// Mitsubishi GX Works2 project: AUTOROLLING_3073_6_2_2026   PLC: Q06UDV
// AUTOROLLING_3073_6_2_2024

PROGRAM 01
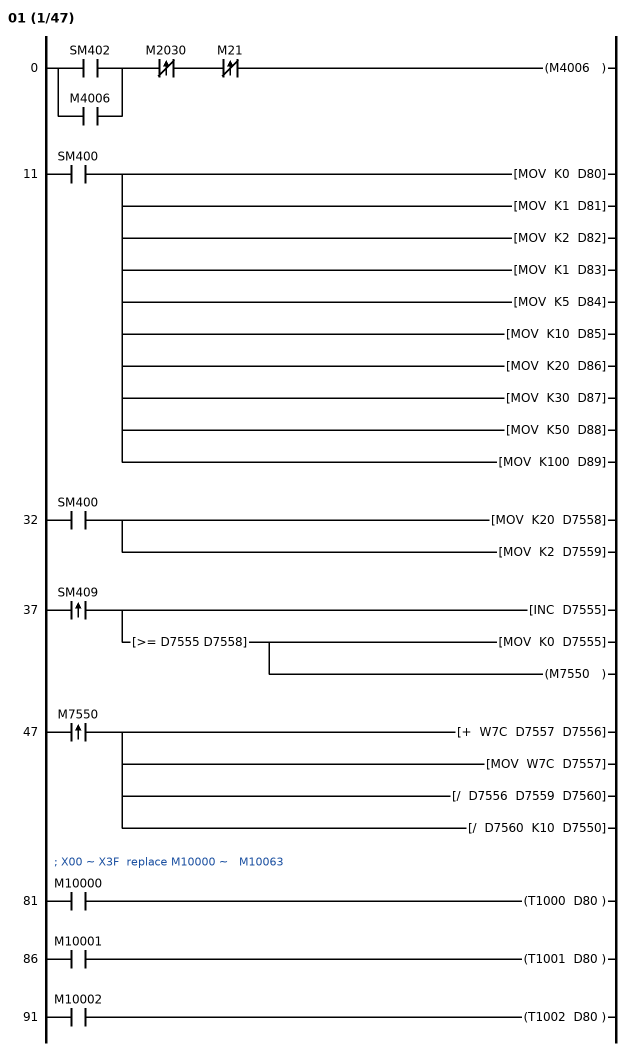
0     LD      SM402
      OR      M4006
      ANDPI   M2030
      ANDPI   M21
      OUT     M4006
; 
; 
; 
11    LD      SM400
      MOV     K0 D80
      MOV     K1 D81
      MOV     K2 D82
      MOV     K1 D83
      MOV     K5 D84
      MOV     K10 D85
      MOV     K20 D86
      MOV     K30 D87
      MOV     K50 D88
      MOV     K100 D89
32    LD      SM400
      MOV     K20 D7558
      MOV     K2 D7559
37    LDP     SM409
      INC     D7555
      AND>=   D7555 D7558
      MOV     K0 D7555
      OUT     M7550
47    LDP     M7550
      +       W7C D7557 D7556
      MOV     W7C D7557
      /       D7556 D7559 D7560
      /       D7560 K10 D7550
; X00 ~ X3F  replace M10000 ~　M10063
81    LD      M10000
      OUT     T1000 D80
86    LD      M10001
      OUT     T1001 D80
91    LD      M10002
      OUT     T1002 D80
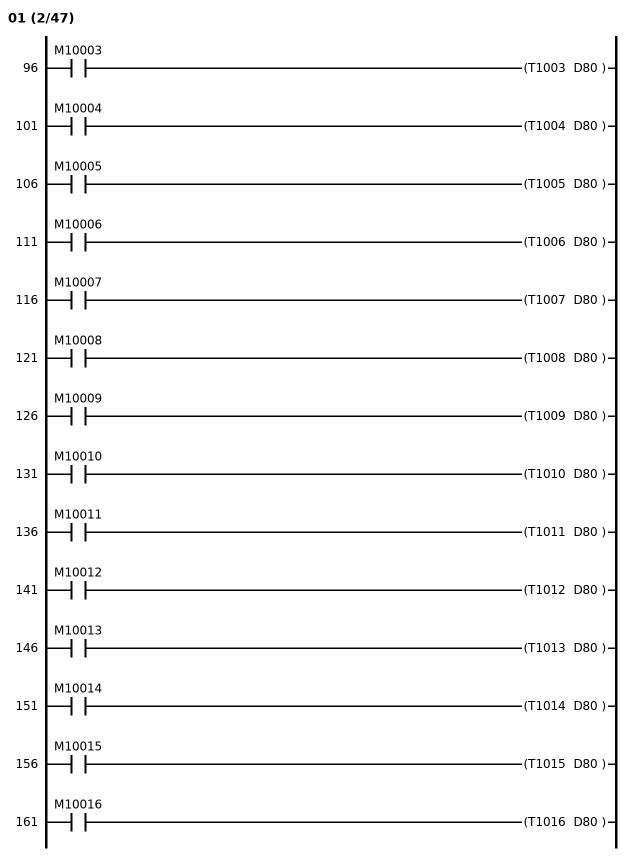
96    LD      M10003
      OUT     T1003 D80
101   LD      M10004
      OUT     T1004 D80
106   LD      M10005
      OUT     T1005 D80
111   LD      M10006
      OUT     T1006 D80
116   LD      M10007
      OUT     T1007 D80
121   LD      M10008
      OUT     T1008 D80
126   LD      M10009
      OUT     T1009 D80
131   LD      M10010
      OUT     T1010 D80
136   LD      M10011
      OUT     T1011 D80
141   LD      M10012
      OUT     T1012 D80
146   LD      M10013
      OUT     T1013 D80
151   LD      M10014
      OUT     T1014 D80
156   LD      M10015
      OUT     T1015 D80
161   LD      M10016
      OUT     T1016 D80
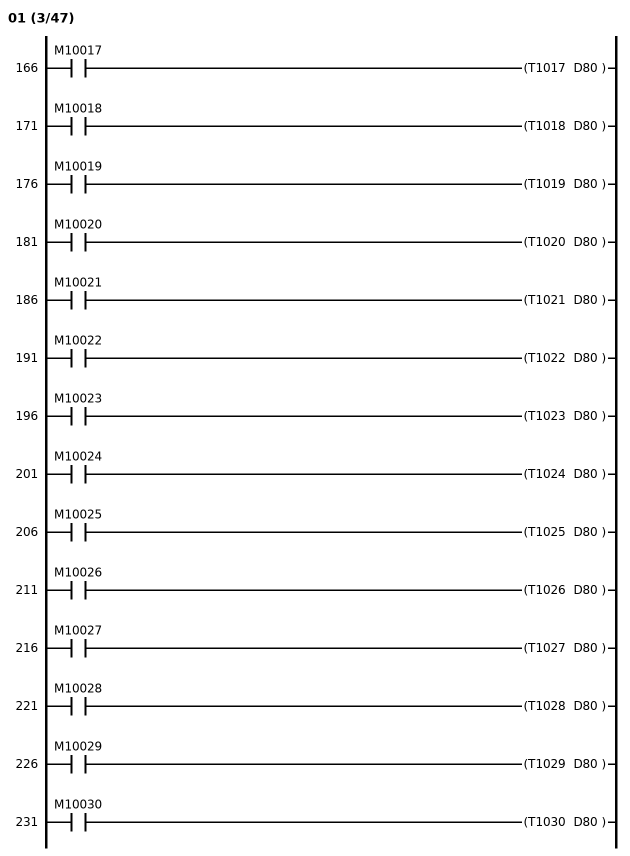
166   LD      M10017
      OUT     T1017 D80
171   LD      M10018
      OUT     T1018 D80
176   LD      M10019
      OUT     T1019 D80
181   LD      M10020
      OUT     T1020 D80
186   LD      M10021
      OUT     T1021 D80
191   LD      M10022
      OUT     T1022 D80
196   LD      M10023
      OUT     T1023 D80
201   LD      M10024
      OUT     T1024 D80
206   LD      M10025
      OUT     T1025 D80
211   LD      M10026
      OUT     T1026 D80
216   LD      M10027
      OUT     T1027 D80
221   LD      M10028
      OUT     T1028 D80
226   LD      M10029
      OUT     T1029 D80
231   LD      M10030
      OUT     T1030 D80
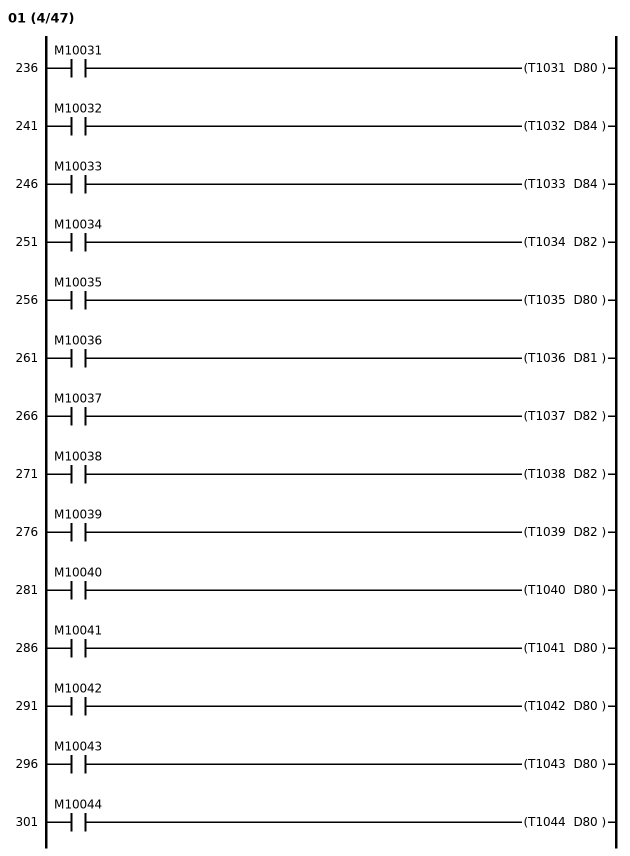
236   LD      M10031
      OUT     T1031 D80
241   LD      M10032
      OUT     T1032 D84
246   LD      M10033
      OUT     T1033 D84
251   LD      M10034
      OUT     T1034 D82
256   LD      M10035
      OUT     T1035 D80
261   LD      M10036
      OUT     T1036 D81
266   LD      M10037
      OUT     T1037 D82
271   LD      M10038
      OUT     T1038 D82
276   LD      M10039
      OUT     T1039 D82
281   LD      M10040
      OUT     T1040 D80
286   LD      M10041
      OUT     T1041 D80
291   LD      M10042
      OUT     T1042 D80
296   LD      M10043
      OUT     T1043 D80
301   LD      M10044
      OUT     T1044 D80
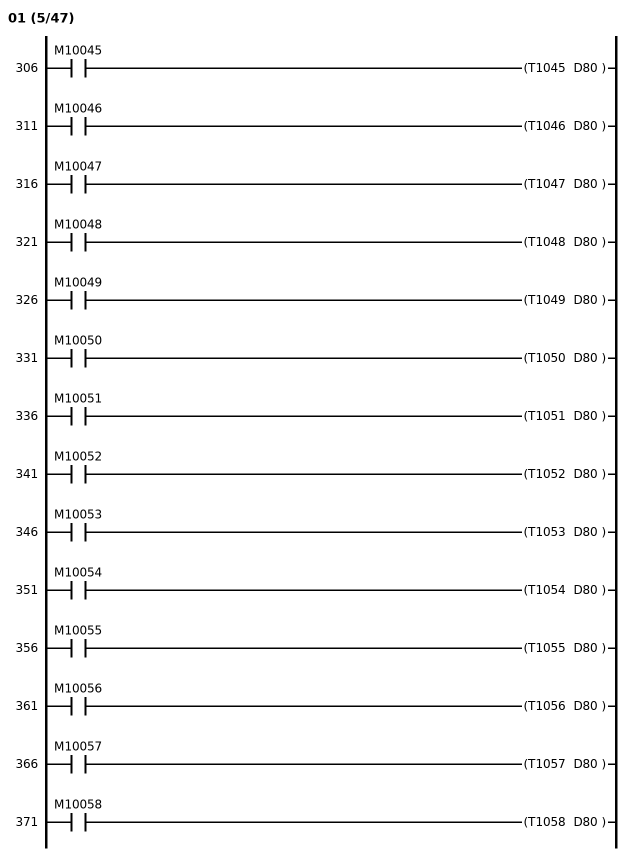
306   LD      M10045
      OUT     T1045 D80
311   LD      M10046
      OUT     T1046 D80
316   LD      M10047
      OUT     T1047 D80
321   LD      M10048
      OUT     T1048 D80
326   LD      M10049
      OUT     T1049 D80
331   LD      M10050
      OUT     T1050 D80
336   LD      M10051
      OUT     T1051 D80
341   LD      M10052
      OUT     T1052 D80
346   LD      M10053
      OUT     T1053 D80
351   LD      M10054
      OUT     T1054 D80
356   LD      M10055
      OUT     T1055 D80
361   LD      M10056
      OUT     T1056 D80
366   LD      M10057
      OUT     T1057 D80
371   LD      M10058
      OUT     T1058 D80
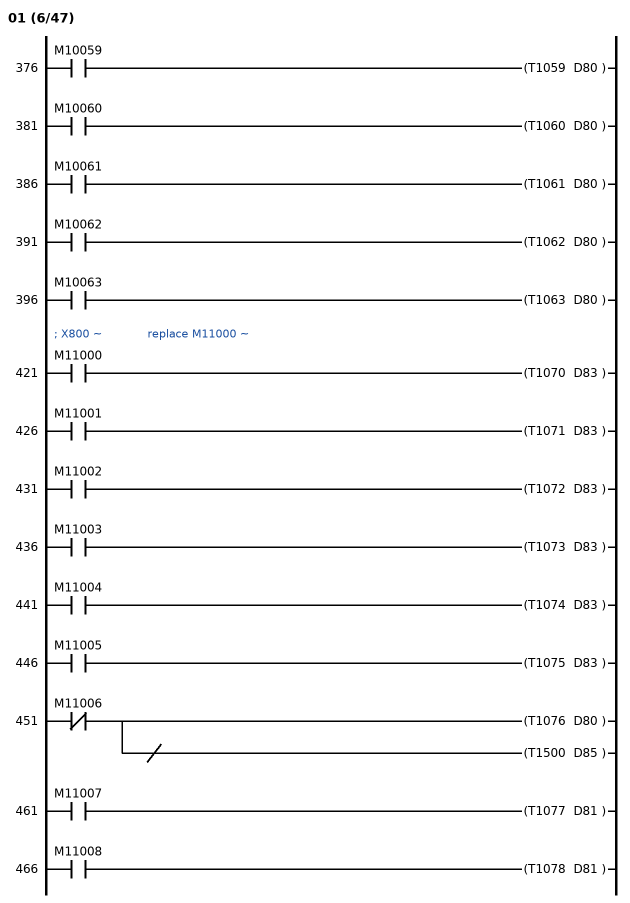
376   LD      M10059
      OUT     T1059 D80
381   LD      M10060
      OUT     T1060 D80
386   LD      M10061
      OUT     T1061 D80
391   LD      M10062
      OUT     T1062 D80
396   LD      M10063
      OUT     T1063 D80
; X800 ~             replace M11000 ~
421   LD      M11000
      OUT     T1070 D83
426   LD      M11001
      OUT     T1071 D83
431   LD      M11002
      OUT     T1072 D83
436   LD      M11003
      OUT     T1073 D83
441   LD      M11004
      OUT     T1074 D83
446   LD      M11005
      OUT     T1075 D83
451   LDI     M11006
      OUT     T1076 D80
      INV
      OUT     T1500 D85
461   LD      M11007
      OUT     T1077 D81
466   LD      M11008
      OUT     T1078 D81
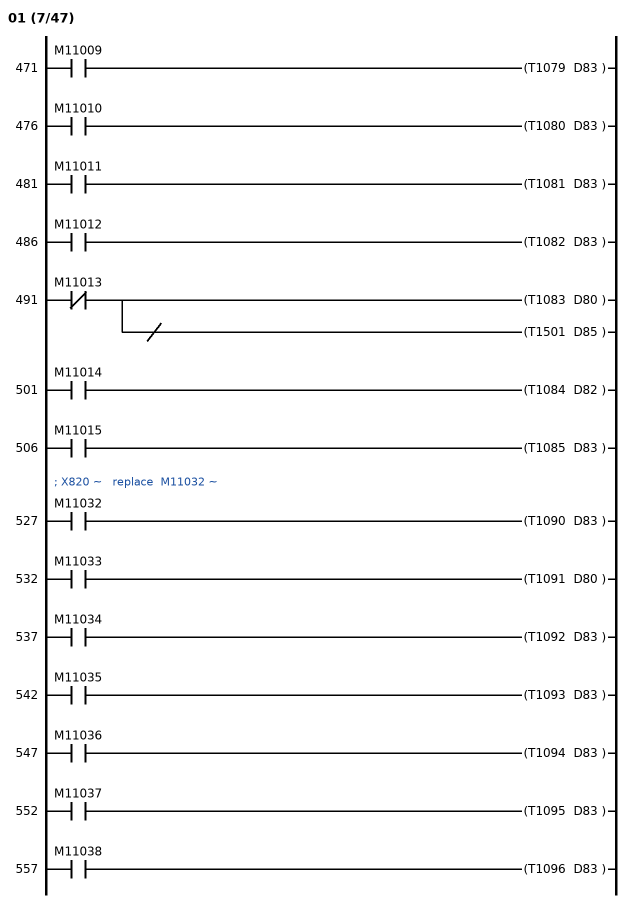
471   LD      M11009
      OUT     T1079 D83
476   LD      M11010
      OUT     T1080 D83
481   LD      M11011
      OUT     T1081 D83
486   LD      M11012
      OUT     T1082 D83
491   LDI     M11013
      OUT     T1083 D80
      INV
      OUT     T1501 D85
501   LD      M11014
      OUT     T1084 D82
506   LD      M11015
      OUT     T1085 D83
; X820 ~   replace  M11032 ~
527   LD      M11032
      OUT     T1090 D83
532   LD      M11033
      OUT     T1091 D80
537   LD      M11034
      OUT     T1092 D83
542   LD      M11035
      OUT     T1093 D83
547   LD      M11036
      OUT     T1094 D83
552   LD      M11037
      OUT     T1095 D83
557   LD      M11038
      OUT     T1096 D83
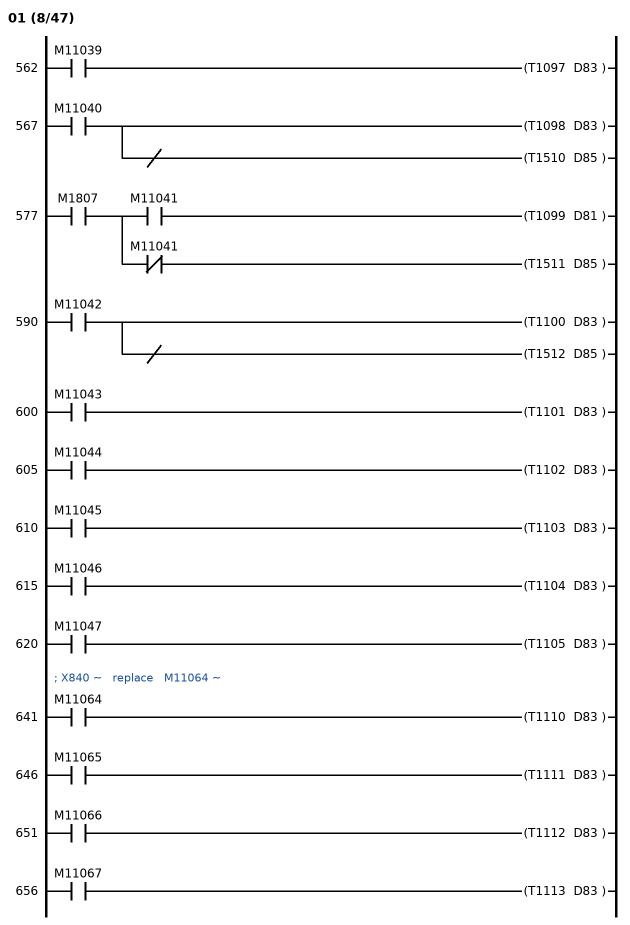
562   LD      M11039
      OUT     T1097 D83
567   LD      M11040
      OUT     T1098 D83
      INV
      OUT     T1510 D85
577   LD      M1807
      MPS
      AND     M11041
      OUT     T1099 D81
      MPP
      ANI     M11041
      OUT     T1511 D85
590   LD      M11042
      OUT     T1100 D83
      INV
      OUT     T1512 D85
600   LD      M11043
      OUT     T1101 D83
605   LD      M11044
      OUT     T1102 D83
610   LD      M11045
      OUT     T1103 D83
615   LD      M11046
      OUT     T1104 D83
620   LD      M11047
      OUT     T1105 D83
; X840 ~   replace   M11064 ~
641   LD      M11064
      OUT     T1110 D83
646   LD      M11065
      OUT     T1111 D83
651   LD      M11066
      OUT     T1112 D83
656   LD      M11067
      OUT     T1113 D83
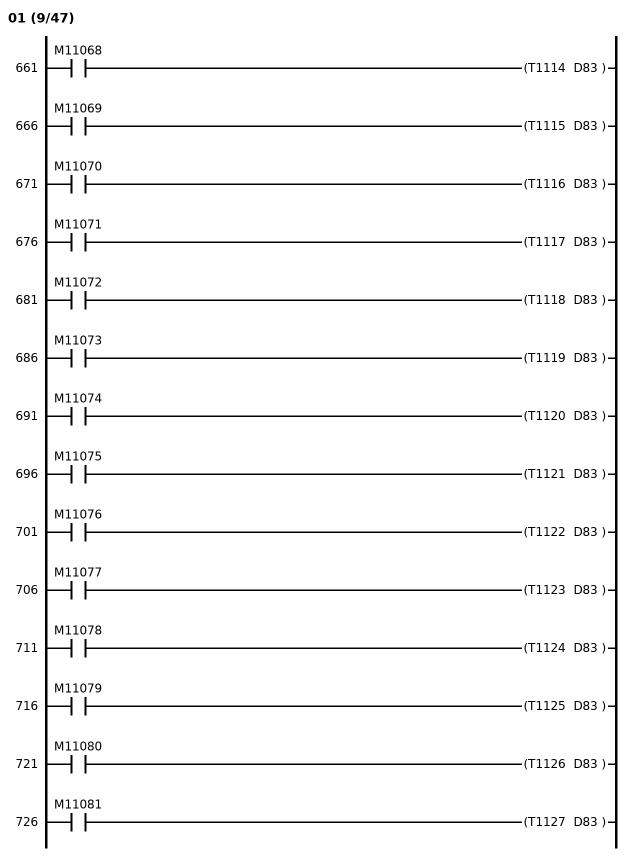
661   LD      M11068
      OUT     T1114 D83
666   LD      M11069
      OUT     T1115 D83
671   LD      M11070
      OUT     T1116 D83
676   LD      M11071
      OUT     T1117 D83
681   LD      M11072
      OUT     T1118 D83
686   LD      M11073
      OUT     T1119 D83
691   LD      M11074
      OUT     T1120 D83
696   LD      M11075
      OUT     T1121 D83
701   LD      M11076
      OUT     T1122 D83
706   LD      M11077
      OUT     T1123 D83
711   LD      M11078
      OUT     T1124 D83
716   LD      M11079
      OUT     T1125 D83
721   LD      M11080
      OUT     T1126 D83
726   LD      M11081
      OUT     T1127 D83
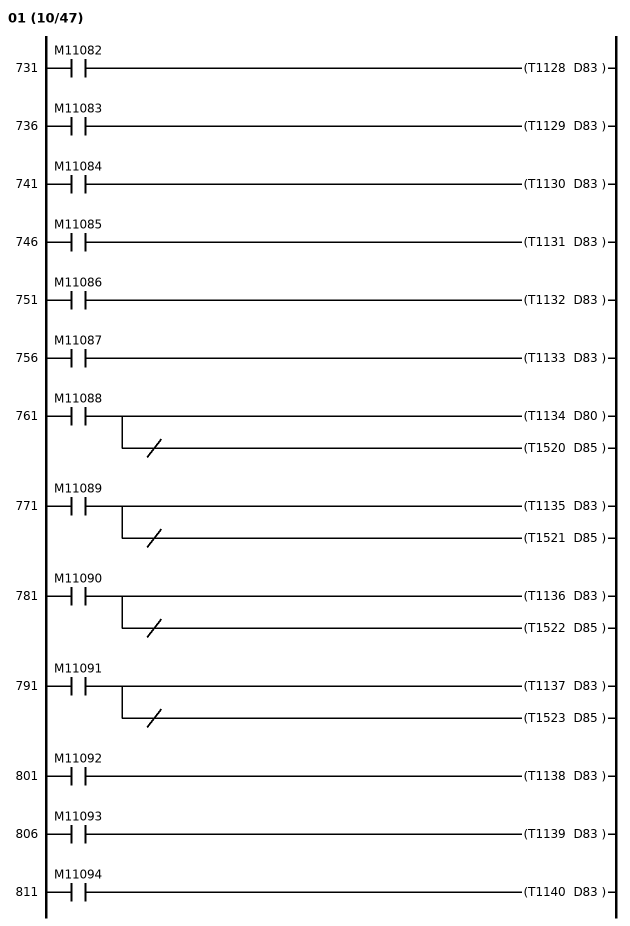
731   LD      M11082
      OUT     T1128 D83
736   LD      M11083
      OUT     T1129 D83
741   LD      M11084
      OUT     T1130 D83
746   LD      M11085
      OUT     T1131 D83
751   LD      M11086
      OUT     T1132 D83
756   LD      M11087
      OUT     T1133 D83
761   LD      M11088
      OUT     T1134 D80
      INV
      OUT     T1520 D85
771   LD      M11089
      OUT     T1135 D83
      INV
      OUT     T1521 D85
781   LD      M11090
      OUT     T1136 D83
      INV
      OUT     T1522 D85
791   LD      M11091
      OUT     T1137 D83
      INV
      OUT     T1523 D85
801   LD      M11092
      OUT     T1138 D83
806   LD      M11093
      OUT     T1139 D83
811   LD      M11094
      OUT     T1140 D83
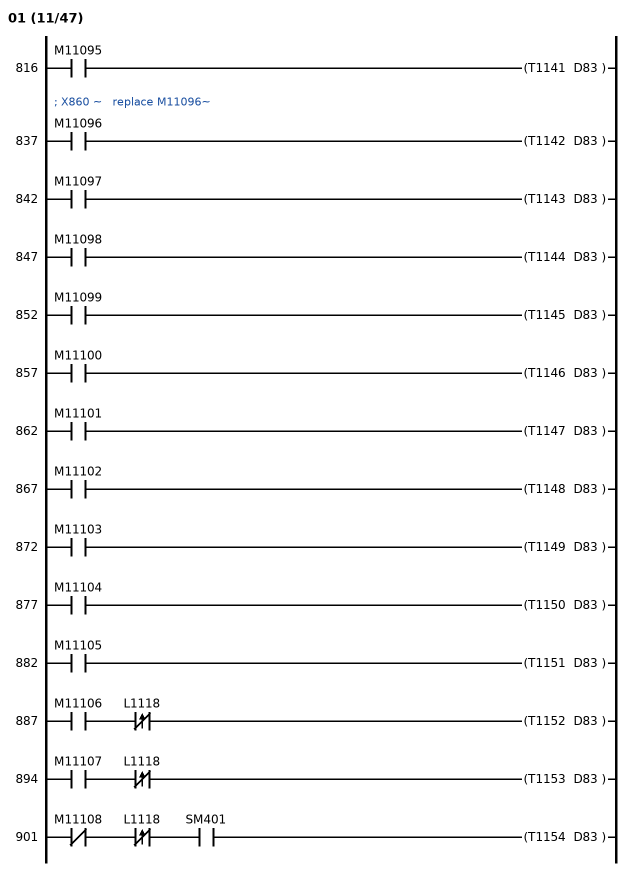
816   LD      M11095
      OUT     T1141 D83
; X860 ~   replace M11096~
837   LD      M11096
      OUT     T1142 D83
842   LD      M11097
      OUT     T1143 D83
847   LD      M11098
      OUT     T1144 D83
852   LD      M11099
      OUT     T1145 D83
857   LD      M11100
      OUT     T1146 D83
862   LD      M11101
      OUT     T1147 D83
867   LD      M11102
      OUT     T1148 D83
872   LD      M11103
      OUT     T1149 D83
877   LD      M11104
      OUT     T1150 D83
882   LD      M11105
      OUT     T1151 D83
887   LD      M11106
      ANDPI   L1118
      OUT     T1152 D83
894   LD      M11107
      ANDPI   L1118
      OUT     T1153 D83
901   LDI     M11108
      ANDPI   L1118
      AND     SM401
      OUT     T1154 D83
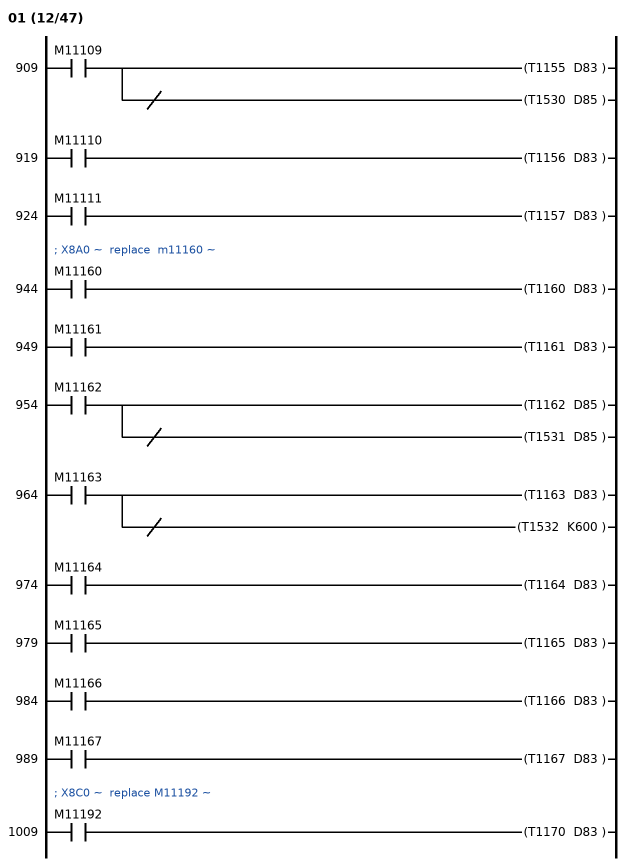
909   LD      M11109
      OUT     T1155 D83
      INV
      OUT     T1530 D85
919   LD      M11110
      OUT     T1156 D83
924   LD      M11111
      OUT     T1157 D83
; X8A0 ~  replace  m11160 ~
944   LD      M11160
      OUT     T1160 D83
949   LD      M11161
      OUT     T1161 D83
954   LD      M11162
      OUT     T1162 D85
      INV
      OUT     T1531 D85
964   LD      M11163
      OUT     T1163 D83
      INV
      OUT     T1532 K600
974   LD      M11164
      OUT     T1164 D83
979   LD      M11165
      OUT     T1165 D83
984   LD      M11166
      OUT     T1166 D83
989   LD      M11167
      OUT     T1167 D83
; X8C0 ~  replace M11192 ~
1009  LD      M11192
      OUT     T1170 D83
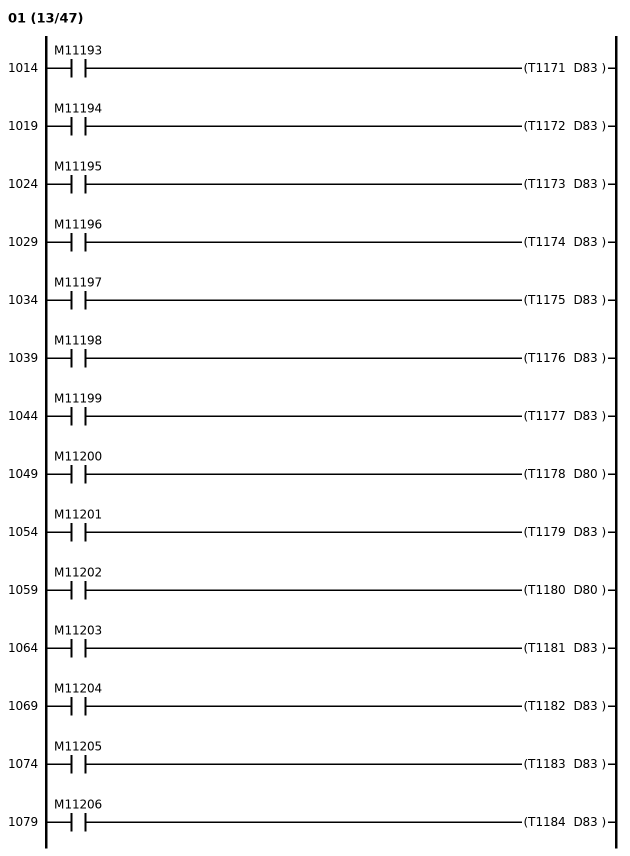
1014  LD      M11193
      OUT     T1171 D83
1019  LD      M11194
      OUT     T1172 D83
1024  LD      M11195
      OUT     T1173 D83
1029  LD      M11196
      OUT     T1174 D83
1034  LD      M11197
      OUT     T1175 D83
1039  LD      M11198
      OUT     T1176 D83
1044  LD      M11199
      OUT     T1177 D83
1049  LD      M11200
      OUT     T1178 D80
1054  LD      M11201
      OUT     T1179 D83
1059  LD      M11202
      OUT     T1180 D80
1064  LD      M11203
      OUT     T1181 D83
1069  LD      M11204
      OUT     T1182 D83
1074  LD      M11205
      OUT     T1183 D83
1079  LD      M11206
      OUT     T1184 D83
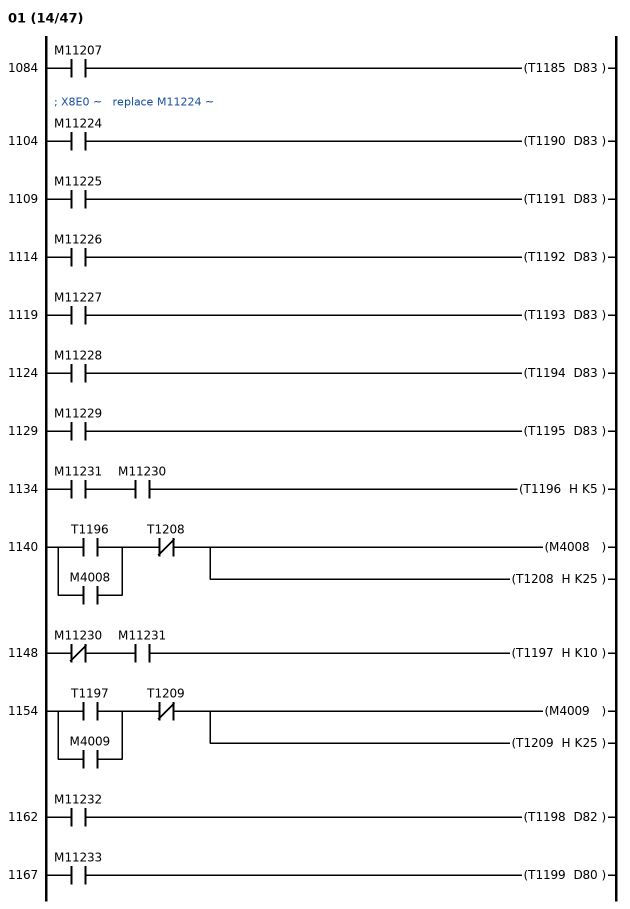
1084  LD      M11207
      OUT     T1185 D83
; X8E0 ~   replace M11224 ~
1104  LD      M11224
      OUT     T1190 D83
1109  LD      M11225
      OUT     T1191 D83
1114  LD      M11226
      OUT     T1192 D83
1119  LD      M11227
      OUT     T1193 D83
1124  LD      M11228
      OUT     T1194 D83
1129  LD      M11229
      OUT     T1195 D83
1134  LD      M11231
      AND     M11230
      OUTH    T1196 K5
1140  LD      T1196
      OR      M4008
      ANI     T1208
      OUT     M4008
      OUTH    T1208 K25
1148  LDI     M11230
      AND     M11231
      OUTH    T1197 K10
1154  LD      T1197
      OR      M4009
      ANI     T1209
      OUT     M4009
      OUTH    T1209 K25
1162  LD      M11232
      OUT     T1198 D82
1167  LD      M11233
      OUT     T1199 D80
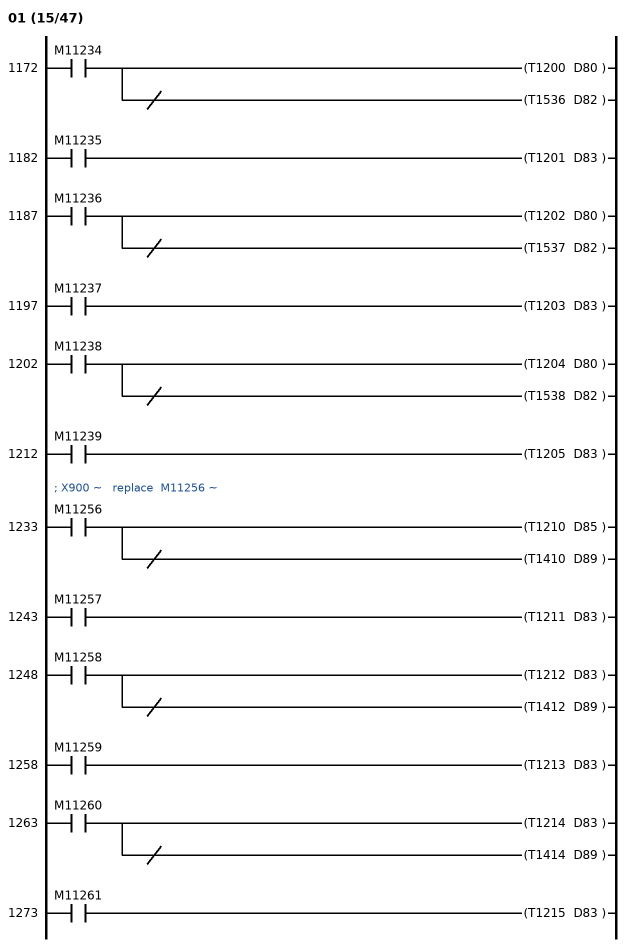
1172  LD      M11234
      OUT     T1200 D80
      INV
      OUT     T1536 D82
1182  LD      M11235
      OUT     T1201 D83
1187  LD      M11236
      OUT     T1202 D80
      INV
      OUT     T1537 D82
1197  LD      M11237
      OUT     T1203 D83
1202  LD      M11238
      OUT     T1204 D80
      INV
      OUT     T1538 D82
1212  LD      M11239
      OUT     T1205 D83
; X900 ~   replace  M11256 ~
1233  LD      M11256
      OUT     T1210 D85
      INV
      OUT     T1410 D89
1243  LD      M11257
      OUT     T1211 D83
1248  LD      M11258
      OUT     T1212 D83
      INV
      OUT     T1412 D89
1258  LD      M11259
      OUT     T1213 D83
1263  LD      M11260
      OUT     T1214 D83
      INV
      OUT     T1414 D89
1273  LD      M11261
      OUT     T1215 D83
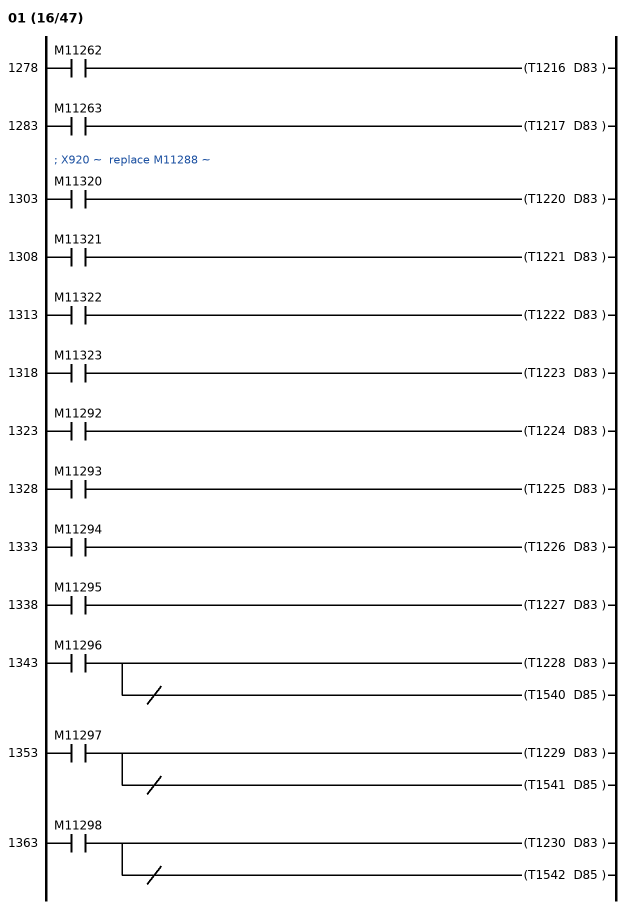
1278  LD      M11262
      OUT     T1216 D83
1283  LD      M11263
      OUT     T1217 D83
; X920 ~  replace M11288 ~
1303  LD      M11320
      OUT     T1220 D83
1308  LD      M11321
      OUT     T1221 D83
1313  LD      M11322
      OUT     T1222 D83
1318  LD      M11323
      OUT     T1223 D83
1323  LD      M11292
      OUT     T1224 D83
1328  LD      M11293
      OUT     T1225 D83
1333  LD      M11294
      OUT     T1226 D83
1338  LD      M11295
      OUT     T1227 D83
1343  LD      M11296
      OUT     T1228 D83
      INV
      OUT     T1540 D85
1353  LD      M11297
      OUT     T1229 D83
      INV
      OUT     T1541 D85
1363  LD      M11298
      OUT     T1230 D83
      INV
      OUT     T1542 D85
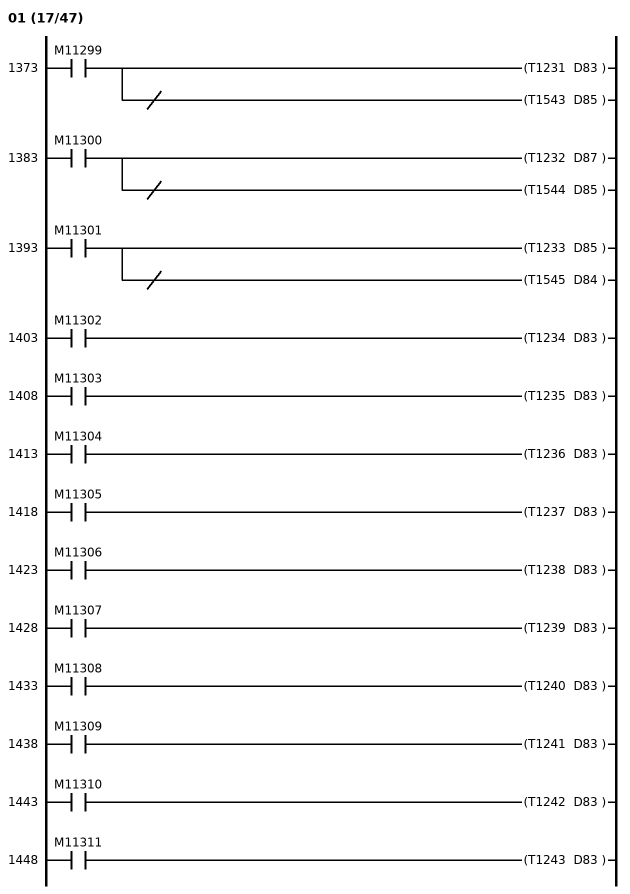
1373  LD      M11299
      OUT     T1231 D83
      INV
      OUT     T1543 D85
1383  LD      M11300
      OUT     T1232 D87
      INV
      OUT     T1544 D85
1393  LD      M11301
      OUT     T1233 D85
      INV
      OUT     T1545 D84
1403  LD      M11302
      OUT     T1234 D83
1408  LD      M11303
      OUT     T1235 D83
1413  LD      M11304
      OUT     T1236 D83
1418  LD      M11305
      OUT     T1237 D83
1423  LD      M11306
      OUT     T1238 D83
1428  LD      M11307
      OUT     T1239 D83
1433  LD      M11308
      OUT     T1240 D83
1438  LD      M11309
      OUT     T1241 D83
1443  LD      M11310
      OUT     T1242 D83
1448  LD      M11311
      OUT     T1243 D83
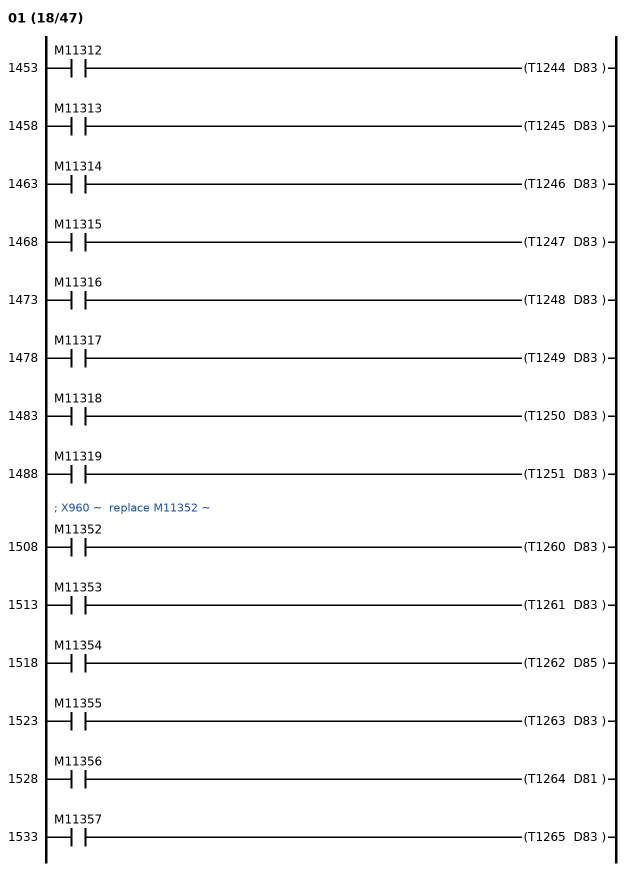
1453  LD      M11312
      OUT     T1244 D83
1458  LD      M11313
      OUT     T1245 D83
1463  LD      M11314
      OUT     T1246 D83
1468  LD      M11315
      OUT     T1247 D83
1473  LD      M11316
      OUT     T1248 D83
1478  LD      M11317
      OUT     T1249 D83
1483  LD      M11318
      OUT     T1250 D83
1488  LD      M11319
      OUT     T1251 D83
; X960 ~  replace M11352 ~
1508  LD      M11352
      OUT     T1260 D83
1513  LD      M11353
      OUT     T1261 D83
1518  LD      M11354
      OUT     T1262 D85
1523  LD      M11355
      OUT     T1263 D83
1528  LD      M11356
      OUT     T1264 D81
1533  LD      M11357
      OUT     T1265 D83
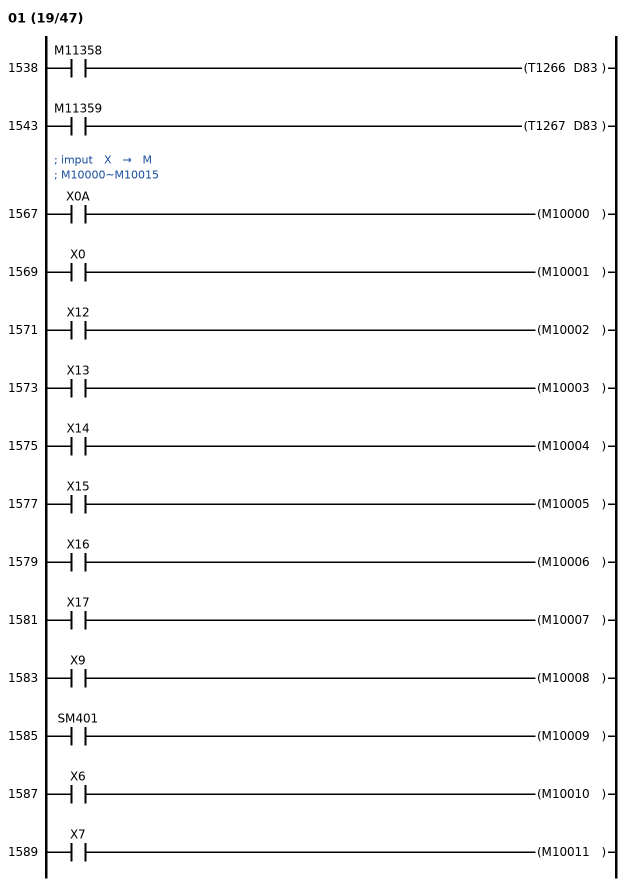
1538  LD      M11358
      OUT     T1266 D83
1543  LD      M11359
      OUT     T1267 D83
; imput　X　→　M
; M10000~M10015
1567  LD      X0A
      OUT     M10000
1569  LD      X0
      OUT     M10001
1571  LD      X12
      OUT     M10002
1573  LD      X13
      OUT     M10003
1575  LD      X14
      OUT     M10004
1577  LD      X15
      OUT     M10005
1579  LD      X16
      OUT     M10006
1581  LD      X17
      OUT     M10007
1583  LD      X9
      OUT     M10008
1585  LD      SM401
      OUT     M10009
1587  LD      X6
      OUT     M10010
1589  LD      X7
      OUT     M10011
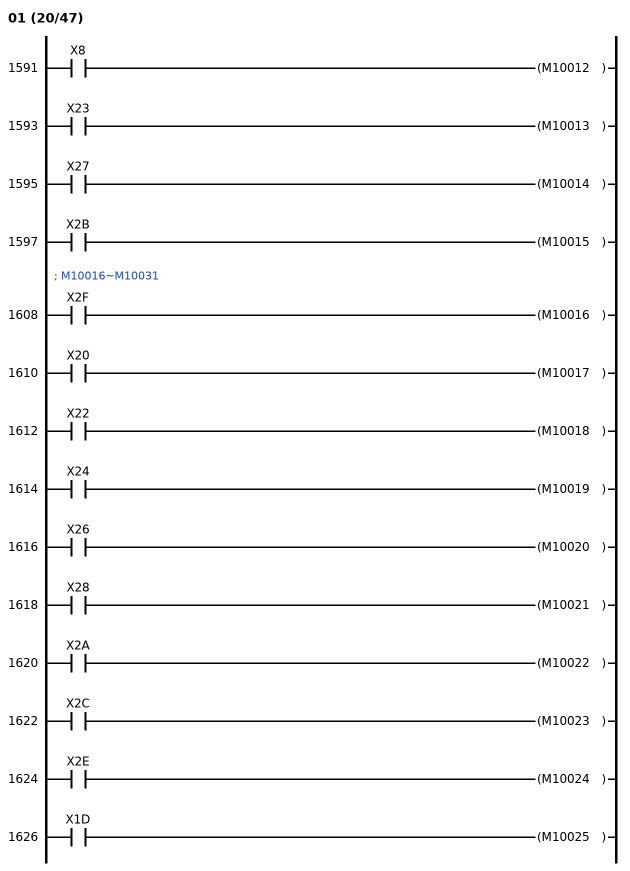
1591  LD      X8
      OUT     M10012
1593  LD      X23
      OUT     M10013
1595  LD      X27
      OUT     M10014
1597  LD      X2B
      OUT     M10015
; M10016~M10031
1608  LD      X2F
      OUT     M10016
1610  LD      X20
      OUT     M10017
1612  LD      X22
      OUT     M10018
1614  LD      X24
      OUT     M10019
1616  LD      X26
      OUT     M10020
1618  LD      X28
      OUT     M10021
1620  LD      X2A
      OUT     M10022
1622  LD      X2C
      OUT     M10023
1624  LD      X2E
      OUT     M10024
1626  LD      X1D
      OUT     M10025
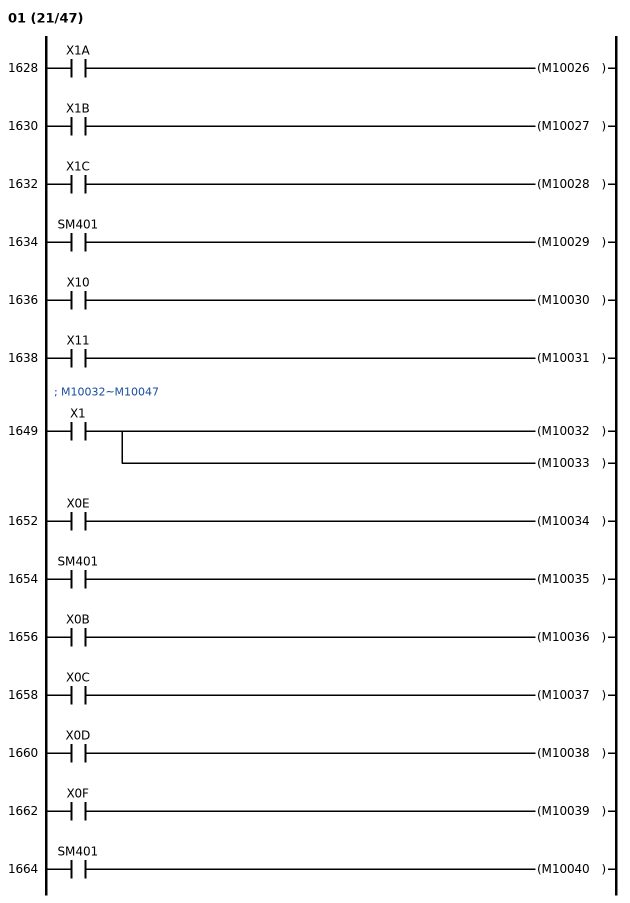
1628  LD      X1A
      OUT     M10026
1630  LD      X1B
      OUT     M10027
1632  LD      X1C
      OUT     M10028
1634  LD      SM401
      OUT     M10029
1636  LD      X10
      OUT     M10030
1638  LD      X11
      OUT     M10031
; M10032~M10047
1649  LD      X1
      OUT     M10032
      OUT     M10033
1652  LD      X0E
      OUT     M10034
1654  LD      SM401
      OUT     M10035
1656  LD      X0B
      OUT     M10036
1658  LD      X0C
      OUT     M10037
1660  LD      X0D
      OUT     M10038
1662  LD      X0F
      OUT     M10039
1664  LD      SM401
      OUT     M10040
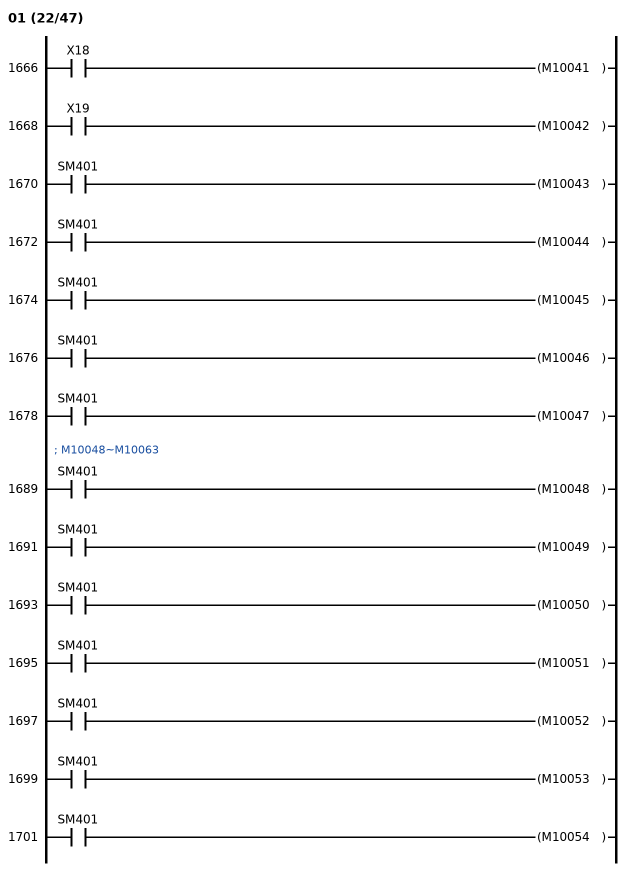
1666  LD      X18
      OUT     M10041
1668  LD      X19
      OUT     M10042
1670  LD      SM401
      OUT     M10043
1672  LD      SM401
      OUT     M10044
1674  LD      SM401
      OUT     M10045
1676  LD      SM401
      OUT     M10046
1678  LD      SM401
      OUT     M10047
; M10048~M10063
1689  LD      SM401
      OUT     M10048
1691  LD      SM401
      OUT     M10049
1693  LD      SM401
      OUT     M10050
1695  LD      SM401
      OUT     M10051
1697  LD      SM401
      OUT     M10052
1699  LD      SM401
      OUT     M10053
1701  LD      SM401
      OUT     M10054
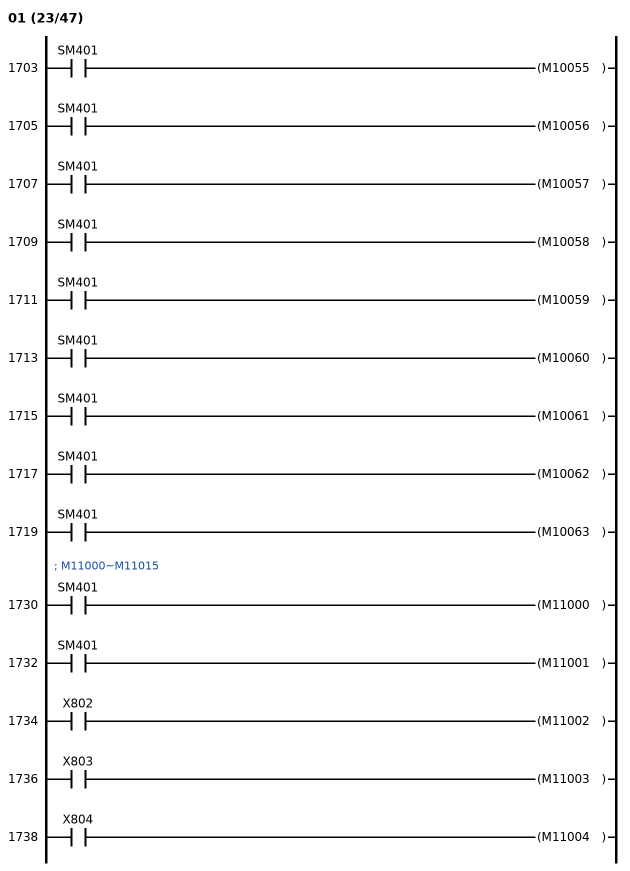
1703  LD      SM401
      OUT     M10055
1705  LD      SM401
      OUT     M10056
1707  LD      SM401
      OUT     M10057
1709  LD      SM401
      OUT     M10058
1711  LD      SM401
      OUT     M10059
1713  LD      SM401
      OUT     M10060
1715  LD      SM401
      OUT     M10061
1717  LD      SM401
      OUT     M10062
1719  LD      SM401
      OUT     M10063
; M11000~M11015
1730  LD      SM401
      OUT     M11000
1732  LD      SM401
      OUT     M11001
1734  LD      X802
      OUT     M11002
1736  LD      X803
      OUT     M11003
1738  LD      X804
      OUT     M11004
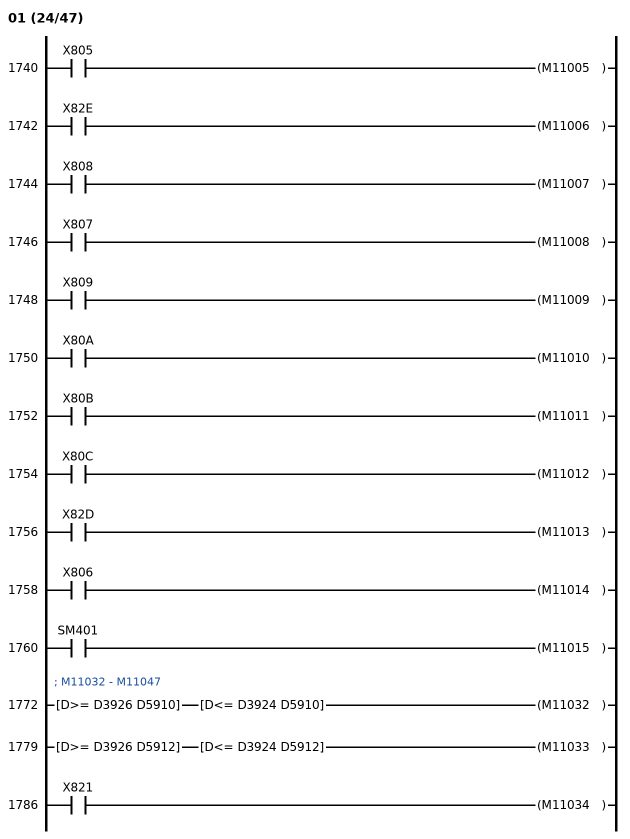
1740  LD      X805
      OUT     M11005
1742  LD      X82E
      OUT     M11006
1744  LD      X808
      OUT     M11007
1746  LD      X807
      OUT     M11008
1748  LD      X809
      OUT     M11009
1750  LD      X80A
      OUT     M11010
1752  LD      X80B
      OUT     M11011
1754  LD      X80C
      OUT     M11012
1756  LD      X82D
      OUT     M11013
1758  LD      X806
      OUT     M11014
1760  LD      SM401
      OUT     M11015
; M11032 - M11047
1772  LDD>=   D3926 D5910
      ANDD<=  D3924 D5910
      OUT     M11032
1779  LDD>=   D3926 D5912
      ANDD<=  D3924 D5912
      OUT     M11033
1786  LD      X821
      OUT     M11034
